(* LS Electric XG5000 project: 2023-09-07 #2 비트연산 *)
(* PLC NewPLC *)
(* module base 0 slot 0: 입력 모듈:XGI-D22A/B (DC 24V 입력, 16점 (전류소스 싱크공용/ 전류소스 입력)) *)
(* module base 0 slot 1: 입력 모듈:XGI-D22A/B (DC 24V 입력, 16점 (전류소스 싱크공용/ 전류소스 입력)) *)
(* module base 0 slot 2: 출력 모듈:XGQ-RY2A/B (릴레이 출력, 16점 (2A용, Varistor 없음/Varistor 부착)) *)
(* module base 0 slot 3: 출력 모듈:XGQ-TR2A/B (트랜지스터 출력, 16점 (0.5A용, 싱크출력/소스출력)) *)
VAR_GLOBAL
    DATA : BYTE;
    PB1 AT P00010 : BIT;
END_VAR

PROGRAM OR연산 (* task: 스캔 프로그램 *)
VAR_EXTERNAL
    DATA : BYTE;
    PB1 : BIT; (* AT P00010 *)
END_VAR

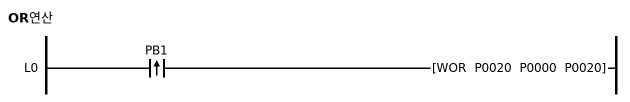
; L0
LOADP     PB1
WOR       P0020 P0000 P0020
END_PROGRAM